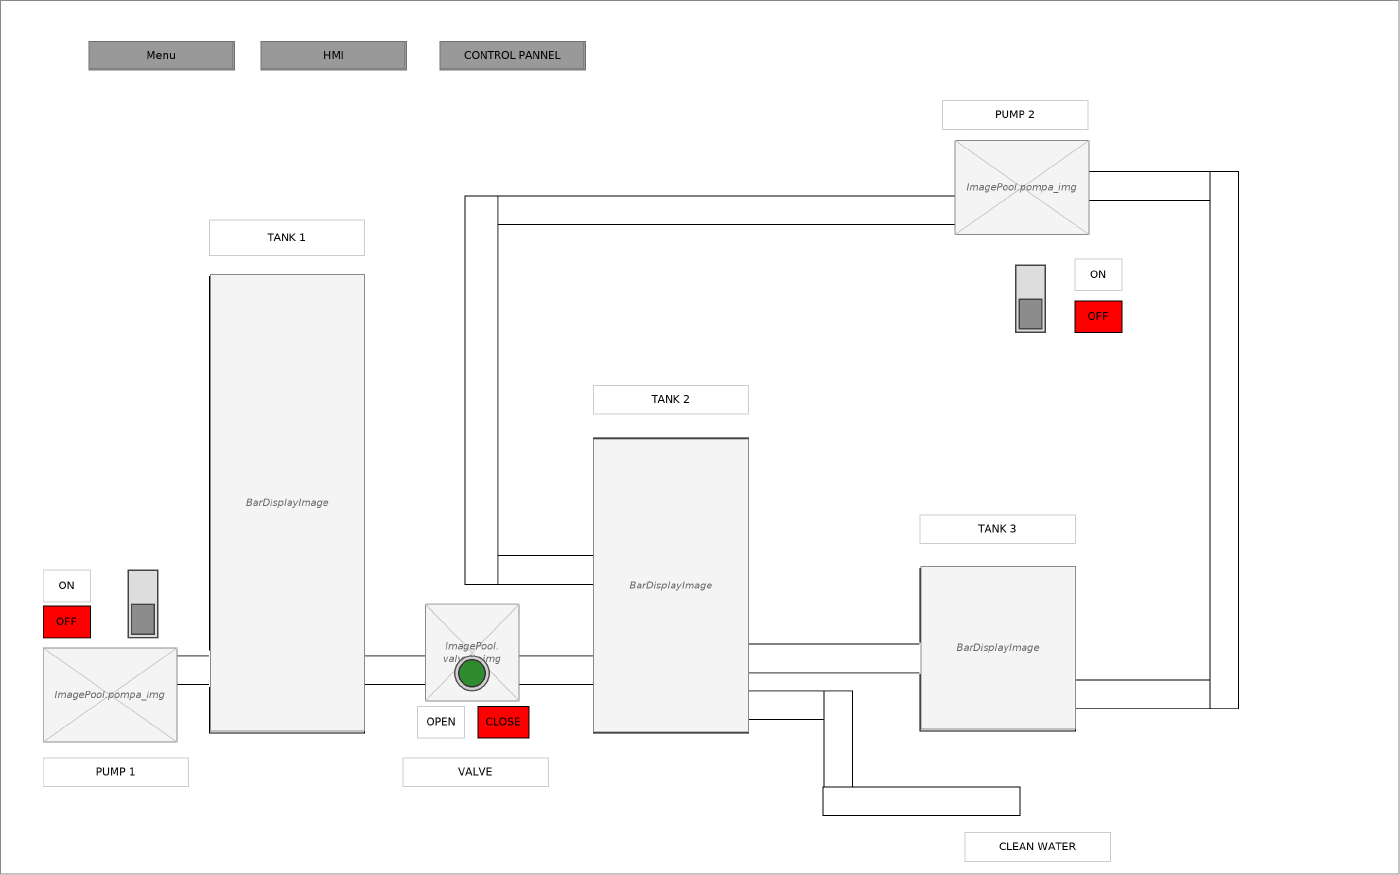
VISUALIZATION Visualization  // 1440x900
    Rectangle (215,284 160x470)
    Rectangle (946,584 160x168)
    Rectangle (610,450 160x304)
    Rectangle (727,662 288x30), colour toggle: HMI.tubeOUT_2
    Rectangle (331,674 354x30), colour toggle: HMI.valve
    Rectangle (145,674 146x30), colour toggle: HMI.pump_1
    Button (91,42 150x30), "Menu"
        OnMouseClick: change screen: Menu
    Button (268,42 150x30), "HMI"
        OnMouseClick: change screen: Visualization
    Button (452,42 150x30), "CONTROL PANNEL"
        OnMouseClick: change screen: Pannello_Controllo
    Textfield (44,779 150x30), "PUMP 1"
    DipSwitch (112,586 70x70), variable: HMI.pump_1, behaviour: TOGGLE, style: Switch-DipSwitch-Gray
    Textfield (44,623 49x33), "OFF", colour toggle: HMI.pump_1
    Textfield (44,586 49x33), "ON", colour toggle: HMI.pump_1
    Textfield (215,226 160x37), "TANK 1"
    Image (44,666 138x97), image: ImagePool.pompa_img
    Textfield (610,396 160x30), "TANK 2"
    Textfield (946,529 160x30), "TANK 3"
    Image (437,621 97x100), image: ImagePool.valvola_img
    Lamp1 (464,669 43x47), variable: HMI.valve, style: Lamp-Lamp1-Green
    Textfield (414,779 150x30), "VALVE"
    Textfield (429,726 49x33), "OPEN", colour toggle: HMI.valve
    Textfield (491,726 53x33), "CLOSE", colour toggle: HMI.valve
    Rectangle (215,669 160x37)
    Rectangle (611,652 158x54)
    BarDisplayImage (216,282 159x470), value: HMI.level_1, style: BarDisplayImage-Gray, scale format: %.1f, scale 0..100
    Rectangle (946,661 90x32)
    Rectangle (759,710 117x30), colour toggle: HMI.tubeOUT_2
    Rectangle (798,759 129x30), angle 90, colour toggle: HMI.tubeOUT_2
    Rectangle (846,809 203x30), colour toggle: HMI.tubeOUT_2
    Textfield (992,856 150x30), "CLEAN WATER"
    Rectangle (726,704 43x37)
    Rectangle (1111,176 162x30), colour toggle: HMI.pump_3
    Rectangle (1095,699 167x30), colour toggle: HMI.pump_3
    DipSwitch (1025,272 70x70), variable: HMI.pump_3, behaviour: TOGGLE, style: Switch-DipSwitch-Gray
    Rectangle (983,437 553x30), angle 90, colour toggle: HMI.pump_3
    Textfield (1105,266 49x33), "ON", colour toggle: HMI.pump_3
    Textfield (1105,309 49x33), "OFF", colour toggle: HMI.pump_3
    Rectangle (984,697 122x32)
    BarDisplayImage (947,582 159x168), value: HMI.level_3, style: BarDisplayImage-Gray, scale format: %.1f, scale 0..4
    Textfield (969,103 150x30), "PUMP 2"
    Rectangle (481,571 211x30), colour toggle: HMI.pump_3
    Rectangle (481,201 511x30), colour toggle: HMI.pump_3
    Rectangle (295,384 400x34), angle 90, colour toggle: HMI.pump_3
    Rectangle (610,570 103x32)
    Image (982,144 138x97), angle 180, image: ImagePool.pompa_img
    BarDisplayImage (610,451 160x302), value: HMI.level_2, style: BarDisplayImage-Gray, scale format: %.1f, scale 0..30
END_VISUALIZATION

(* stored: Version 1.1.0.1
   Visu Visualization: Id {a8246ed9-12a7-45ca-b47e-e2c9ba14f292} *)
